VAR_GLOBAL CONSTANT
	cRECVDATACHANNELBUFFER: INT := 20;
END_VAR

(* stored: Version 1.1.0.1, ProductVersion 3.1.0.25
   GVL OvenConst: Id {72d8bda2-44e8-476b-a778-767834ec8549} *)
